PROGRAM MAIN
VAR
END_VAR

Reservoir();

END_PROGRAM

(* stored: Version 1.1.0.1, ProductVersion 3.1.4024.12
   POU MAIN: Id {2efee629-8525-4c5f-b2a6-bd758d48f9a5}, SpecialFunc None *)
